FUNCTION TryConvert_BOOL_TO_LWORD : BOOL
VAR_INPUT
	in : BOOL;
	out : REFERENCE TO LWORD;
END_VAR

out := BOOL_TO_LWORD(in);
TryConvert_BOOL_TO_LWORD := TRUE;

END_FUNCTION

(* stored: Version 1.1.0.1, ProductVersion 3.1.4024.12
   POU TryConvert_BOOL_TO_LWORD: Id {e361a99e-f650-4dfe-ac62-dfdf170bf6b2}, SpecialFunc None *)
